// TIA Portal V18 export
FUNCTION "F_ChannelDia" : Void   // FC2, F_LAD
{ S7_Optimized_Access := 'TRUE' }
VERSION : 0.1
// stored: AutoNumber true, IsIECCheckEnabled false, UDAEnableTagReadback false
   VAR_INPUT
      PASS_OUT : Bool;
      QBAD : Bool;
      ACK_REQ : Bool;
      Channel0_ValueStatus : Bool;
      Channel1_ValueStatus : Bool;
      Channel2_ValueStatus : Bool;
      Channel3_ValueStatus : Bool;
      Channel4_ValueStatus : Bool;
      Channel5_ValueStatus : Bool;
      Channel6_ValueStatus : Bool;
      Channel7_ValueStatus : Bool;
   END_VAR
   VAR_OUTPUT
      FIODia : "FIODia";
   END_VAR
   VAR_TEMP   // added for the SCL form of the ladder/FBD networks
      _w1 : Bool;
   END_VAR
BEGIN

REGION Network 1: 模块钝化
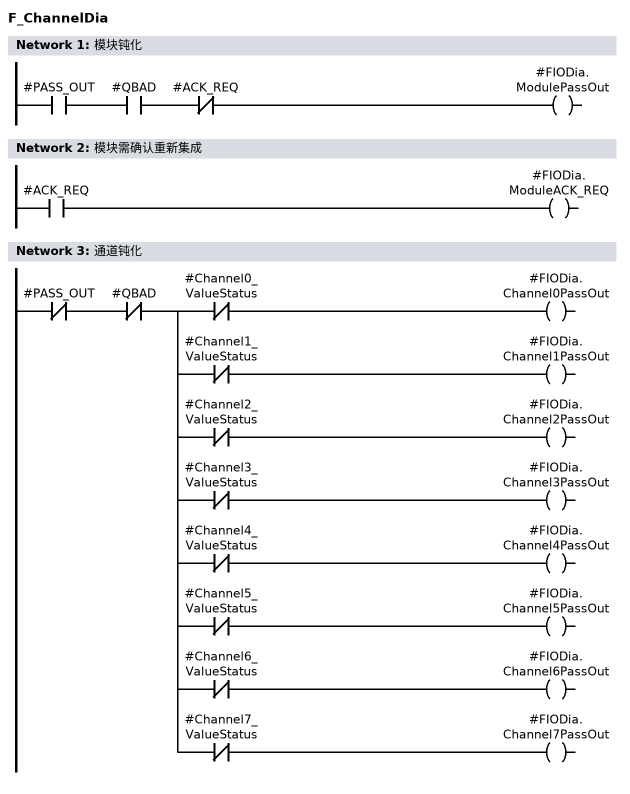
   RUNG wire#powerrail
      Contact( #PASS_OUT )
      Contact( #QBAD )
      I_Contact( #ACK_REQ )
      Coil( #FIODia.ModulePassOut )
   END_RUNG
   // the same network as SCL:
   #FIODia.ModulePassOut := #PASS_OUT AND #QBAD AND NOT #ACK_REQ;
END_REGION

REGION Network 2: 模块需确认重新集成
   RUNG wire#powerrail
      Contact( #ACK_REQ )
      Coil( #FIODia.ModuleACK_REQ )
   END_RUNG
   // the same network as SCL:
   #FIODia.ModuleACK_REQ := #ACK_REQ;
END_REGION

REGION Network 3: 通道钝化
   RUNG wire#powerrail
      I_Contact( #PASS_OUT )
      I_Contact( #QBAD )
      wire#w1
      I_Contact( #Channel0_ValueStatus )
      Coil( #FIODia.Channel0PassOut )
   END_RUNG
   RUNG wire#w1
      I_Contact( #Channel1_ValueStatus )
      Coil( #FIODia.Channel1PassOut )
   END_RUNG
   RUNG wire#w1
      I_Contact( #Channel2_ValueStatus )
      Coil( #FIODia.Channel2PassOut )
   END_RUNG
   RUNG wire#w1
      I_Contact( #Channel3_ValueStatus )
      Coil( #FIODia.Channel3PassOut )
   END_RUNG
   RUNG wire#w1
      I_Contact( #Channel4_ValueStatus )
      Coil( #FIODia.Channel4PassOut )
   END_RUNG
   RUNG wire#w1
      I_Contact( #Channel5_ValueStatus )
      Coil( #FIODia.Channel5PassOut )
   END_RUNG
   RUNG wire#w1
      I_Contact( #Channel6_ValueStatus )
      Coil( #FIODia.Channel6PassOut )
   END_RUNG
   RUNG wire#w1
      I_Contact( #Channel7_ValueStatus )
      Coil( #FIODia.Channel7PassOut )
   END_RUNG
   // the same network as SCL:
   #_w1 := NOT #PASS_OUT AND NOT #QBAD;
   #FIODia.Channel0PassOut := #_w1 AND NOT #Channel0_ValueStatus;
   #FIODia.Channel1PassOut := #_w1 AND NOT #Channel1_ValueStatus;
   #FIODia.Channel2PassOut := #_w1 AND NOT #Channel2_ValueStatus;
   #FIODia.Channel3PassOut := #_w1 AND NOT #Channel3_ValueStatus;
   #FIODia.Channel4PassOut := #_w1 AND NOT #Channel4_ValueStatus;
   #FIODia.Channel5PassOut := #_w1 AND NOT #Channel5_ValueStatus;
   #FIODia.Channel6PassOut := #_w1 AND NOT #Channel6_ValueStatus;
   #FIODia.Channel7PassOut := #_w1 AND NOT #Channel7_ValueStatus;
END_REGION
END_FUNCTION
